TEXTLIST TextListForCombobox_eSignalform
  1 = 'OFF'
  2 = 'OFFSET'
  3 = 'RECHTECK'
  4 = 'DREIECK'
  5 = 'SINUS'
   = ''
END_TEXTLIST

(* stored: Version 1.1.0.1, ProductVersion 3.1.4024.12
   TextList TextListForCombobox_eSignalform: Id {8420a506-94e1-4f11-b163-04c32a093ef7} *)
